FUNCTION_BLOCK PUBLIC EventHandlerInterface_TestSuite EXTENDS TcUnit.FB_TestSuite
VAR
END_VAR

CheckEmitWorksWithHandler();
CheckExtendsFromQueryInterface();

METHOD PUBLIC CheckEmitWorksWithHandler
VAR
	mockEvent : MockEvent;
	mockHandler : MockEventHandler;
	iEventHandler : I_EventHandler := mockHandler;
	eventEmitter : EventEmitter;
	eventReceived : BOOL;
END_VAR
TEST('CheckEmitWorksWithHandler');

eventEmitter.OnEvent('test', iEventHandler);

eventEmitter.Emit('test',mockEvent);
eventReceived := mockHandler.EqualsLastEvent(mockEvent);

AssertTrue(
	Condition := eventReceived,
	Message := 'Event Emitter did not correctly emmit the event to the handler'
);

TEST_FINISHED();
END_METHOD

METHOD PUBLIC CheckExtendsFromQueryInterface
VAR
	mockHandler : MockEventHandler;
	iEventHandler : I_EventHandler := mockHandler;
	iQueryInterface : __SYSTEM.IQueryInterface;
	result : BOOL;
END_VAR
TEST('CheckExtendsFromQueryInterface');

result := __QUERYINTERFACE(iEventHandler,iQueryInterface);

AssertTrue(
	Condition := result,
	Message := 'Interface did not extend __SYSTEM.IQueryInterface'
);

TEST_FINISHED();
END_METHOD

END_FUNCTION_BLOCK

(* stored: Version 1.1.0.1, ProductVersion 3.1.4024.12
   POU EventHandlerInterface_TestSuite: Id {6d96a987-67b0-465f-99b8-e880f93f05a8}, SpecialFunc None
   Method CheckEmitWorksWithHandler: Id {2d70aa61-0631-454d-90ab-1076ce909a5d}
   Method CheckExtendsFromQueryInterface: Id {ffc48322-d2ee-464b-abe4-8e808aba3d98} *)
